FUNCTION F_RAW_TO_PHYS_LREAL (* Convert ISOBUS raw UDINT to physical LREAL value. ISOBUS formula: display = (raw + offset) * scale Example: raw=50000, scale=0.01, offset=-100000 DINT(50000) + (-100000) = -50000 REAL(-50000) 0.01     = -500.0 *)
  (* Standard: 61499-2; Description: Copyright (c) 2026 Meisterschulen am Ostbahnhof This program and the accompanying materials are made available under the terms of the Eclipse Public License 2.0 which is available at https://www.eclipse.org/legal/epl-2.0/ SPDX-License-Identifier: EPL-2.0 *)
  (* Version 1.0, 2026-04-14, Franz Höpfinger, Meisterschulen am Ostbahnhof *)
  PACKAGE logiBUS::utils::conversion::phys;
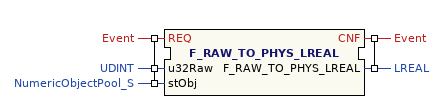
  EVENT_INPUT
    REQ WITH u32Raw, stObj;
  END_EVENT
  EVENT_OUTPUT
    CNF WITH F_RAW_TO_PHYS_LREAL;
  END_EVENT
  VAR_INPUT
    u32Raw : UDINT;
    stObj : logiBUS::utils::conversion::phys::NumericObjectPool_S;
  END_VAR
  VAR_OUTPUT
    F_RAW_TO_PHYS_LREAL : LREAL;
  END_VAR
  BODY IN ST:
PACKAGE logiBUS::utils::conversion::phys;

(* Convert ISOBUS raw UDINT to physical LREAL value.
 * ISOBUS formula: display = (raw + offset) * scale
 * *
 * Example: raw=50000, scale=0.01, offset=-100000 DINT(50000) + (-100000) = -50000 REAL(-50000) *
 * 0.01     = -500.0 *)
FUNCTION F_RAW_TO_PHYS_LREAL : LREAL

VAR_INPUT
	u32Raw : UDINT;
	stObj : NumericObjectPool_S;
END_VAR

VAR_TEMP
	i64Raw : LINT; // to avoid overflow
	i64Offset : LINT; // to avoid overflow
END_VAR

i64Raw := u32Raw; // no conversion needed
i64Offset := stObj.i32Offset; // no conversion needed

F_RAW_TO_PHYS_LREAL := LINT_TO_LREAL(i64Raw + i64Offset) * stObj.r32Scale;

END_FUNCTION
  END_BODY
END_FUNCTION
